(* IEC 61131-3 sources: Word/plc-course/24-capstone-projects/labs/starter, 3 files *)

(* ---- 24-1-conveyor-sorting-cell.st ---- *)
(* Capstone 24-1: Conveyor sorting cell SC-1.
   Module 24 (Capstone projects). STARTER - the interface is done for you.

   Everything the acceptance test (FAT) uses is declared here: the I/O, the
   HMI interface structure and the configuration. Do not rename any of it.
   Everything else is your design. Read the brief first:
     24-capstone-projects/24-1-conveyor-sorting-cell.md

   Suggested workflow:
     1. Add your own types (state enumeration, tracking record, ...) in a
        second TYPE block, and your function blocks (for example FB_Alarm,
        FB_Pusher, FB_Tracker) between the TYPE blocks and the PROGRAM.
     2. Replace the placeholder body of SortingCell with your logic.
     3. Run the FAT and work through it milestone by milestone (M1..M7):
          python3 tools/plctest.py my-work/24-1-conveyor-sorting-cell.st \
                  24-capstone-projects/labs/24-1-conveyor-sorting-cell.test

   Training exercise only. The emergency stop is read here as an ordinary
   input so that the program can react to it. On a real machine the
   emergency stop is a safety function: a safety relay or safety PLC
   removes power from the motor and the pusher valves directly, and the
   standard PLC only monitors it (Module 20). *)

TYPE
  (* ---- HMI interface: part of the specification, do not change ---- *)
  ST_CellCmd : STRUCT            (* HMI -> PLC. The HMI sets a bit, the PLC acts once and clears it *)
    Start        : BOOL;         (* start the cell (Auto) *)
    Stop         : BOOL;         (* normal stop, always obeyed *)
    Ack          : BOOL;         (* acknowledge all alarms *)
    Reset        : BOOL;         (* acknowledge and reset alarms whose cause has gone *)
    CyclePusherA : BOOL;         (* Manual: one supervised stroke of pusher A *)
    CyclePusherB : BOOL;         (* Manual: one supervised stroke of pusher B *)
    ClearCounts  : BOOL;         (* zero all six production counters *)
  END_STRUCT;

  ST_CellSts : STRUCT            (* PLC -> HMI, rewritten every scan *)
    State          : INT;        (* 1 STOPPED, 2 STARTING, 3 RUNNING, 4 FAULTED, 5 MANUAL *)
    Ready          : BOOL;       (* a Start now would be accepted *)
    LaneAFull      : BOOL;       (* debounced lane-full status *)
    LaneBFull      : BOOL;
    PartsInTransit : INT;        (* registered parts not yet delivered *)
    CountMetal     : DINT;       (* classified at the entry station *)
    CountPlastic   : DINT;
    CountOversize  : DINT;
    CountLaneA     : DINT;       (* delivered, counted by the delivery eyes *)
    CountLaneB     : DINT;
    CountReject    : DINT;
  END_STRUCT;

  ST_CellAlm : STRUCT            (* PLC -> HMI. TRUE from detection until a successful reset *)
    EStop         : BOOL;
    MotorOverload : BOOL;
    EntryJam      : BOOL;        (* entry eye blocked too long *)
    Jam           : BOOL;        (* a part did not reach its delivery eye in time *)
    PusherA       : BOOL;        (* pusher A did not extend / retract / stay home *)
    PusherB       : BOOL;
    TrackOverflow : BOOL;        (* more parts on the belt than the tracking table holds *)
    Unacked       : BOOL;        (* at least one alarm not yet acknowledged *)
  END_STRUCT;

  ST_CellCfg : STRUCT            (* engineer settings; the defaults are the commissioning values *)
    StartWarnTime : TIME := T#3s;    (* horn before the belt moves (never less than 2 s) *)
    DistA         : INT  := 500;     (* mm from registration to pusher A *)
    DistB         : INT  := 1000;    (* mm from registration to pusher B *)
    JamTimeA      : TIME := T#3s;    (* running time allowed from registration to LaneA_PE *)
    JamTimeB      : TIME := T#4s;    (* ... to LaneB_PE *)
    JamTimeR      : TIME := T#5s;    (* ... to RejectPE *)
    EntryJamTime  : TIME := T#2s;    (* entry eye blocked while running *)
    PusherTimeout : TIME := T#1s;    (* each pusher movement must finish within this *)
    LaneFullTime  : TIME := T#1s;    (* lane-full eye debounce, on and off *)
  END_STRUCT;

  ST_CellHmi : STRUCT
    Cmd : ST_CellCmd;
    Sts : ST_CellSts;
    Alm : ST_CellAlm;
    Cfg : ST_CellCfg;
  END_STRUCT;
END_TYPE

(* TODO: your own TYPE block and your function blocks go here. *)

PROGRAM SortingCell
  VAR (* operator panel *)
    StartPB    AT %IX0.0 : BOOL;   (* Start, NO *)
    StopPB_NC  AT %IX0.1 : BOOL;   (* Stop, NC: TRUE while not pressed *)
    EStop_NC   AT %IX0.2 : BOOL;   (* e-stop circuit monitoring, NC: TRUE while healthy *)
    ResetPB    AT %IX0.3 : BOOL;   (* Reset, NO *)
    ModeAuto   AT %IX0.4 : BOOL;   (* mode selector in AUTO *)
    ModeManual AT %IX0.5 : BOOL;   (* mode selector in MAN *)
    JogPB      AT %IX0.6 : BOOL;   (* Jog forward, NO, hold-to-run *)
    MotorOL_NC AT %IX0.7 : BOOL;   (* conveyor motor overload relay, NC: TRUE while healthy *)
  END_VAR
  VAR (* conveyor sensors *)
    EntryPE       AT %IX1.0 : BOOL;  (* entry eye: TRUE while a part blocks it *)
    MetalPX       AT %IX1.1 : BOOL;  (* inductive sensor: TRUE = metal *)
    TallPE        AT %IX1.2 : BOOL;  (* height eye: TRUE = part too tall *)
    LaneA_PE      AT %IX1.3 : BOOL;  (* lane A delivery eye *)
    LaneB_PE      AT %IX1.4 : BOOL;  (* lane B delivery eye *)
    RejectPE      AT %IX1.5 : BOOL;  (* reject chute eye *)
    LaneA_FullPE  AT %IX1.6 : BOOL;  (* lane A full eye: TRUE = blocked *)
    LaneB_FullPE  AT %IX1.7 : BOOL;  (* lane B full eye *)
    PusherA_ExtLS AT %IX2.0 : BOOL;  (* pusher A extended *)
    PusherA_RetLS AT %IX2.1 : BOOL;  (* pusher A retracted (home) *)
    PusherB_ExtLS AT %IX2.2 : BOOL;  (* pusher B extended *)
    PusherB_RetLS AT %IX2.3 : BOOL;  (* pusher B retracted (home) *)
    EncCount      AT %IW0 : UINT;    (* belt encoder via high-speed counter: 1 count = 1 mm *)
  END_VAR
  VAR (* outputs *)
    ConveyorRun AT %QX0.0 : BOOL;    (* conveyor motor contactor *)
    PusherA_Sol AT %QX0.1 : BOOL;    (* pusher A solenoid valve: TRUE = extend *)
    PusherB_Sol AT %QX0.2 : BOOL;    (* pusher B solenoid valve *)
    Horn        AT %QX0.3 : BOOL;    (* start-up warning horn *)
    GreenLamp   AT %QX0.4 : BOOL;    (* stack light green: running *)
    AmberLamp   AT %QX0.5 : BOOL;    (* stack light amber: lane full *)
    RedLamp     AT %QX0.6 : BOOL;    (* stack light red: alarm *)
  END_VAR
  VAR (* HMI interface *)
    HMI : ST_CellHmi;
  END_VAR
  (* TODO: your internal variables and function block instances. *)

  (* TODO: replace these placeholder lines with the cell logic.
     (MATIEC needs at least one statement in a program body.) *)
  ConveyorRun := FALSE;
  PusherA_Sol := FALSE;
  PusherB_Sol := FALSE;
  Horn := FALSE;
  GreenLamp := FALSE;
  AmberLamp := FALSE;
  RedLamp := FALSE;
  HMI.Sts.State := 1;
END_PROGRAM

CONFIGURATION Config0
  RESOURCE Res0 ON PLC
    TASK MainTask(INTERVAL := T#10ms, PRIORITY := 0);
    PROGRAM Inst0 WITH MainTask : SortingCell;
  END_RESOURCE
END_CONFIGURATION

(* ---- 24-2-batch-mixing-plant.st ---- *)
(* Capstone 24-2: Batch mixing plant (mixing vessel T-201).
   Module 24 (Capstone projects). STARTER - the interface, the recipe,
   configuration, HMI and report data types, and the plant simulation are
   done for you. Write the control logic where it says TODO (add your own
   functions, function blocks and variables as you wish), then run:
     python3 tools/plctest.py 24-capstone-projects/labs/starter/24-2-batch-mixing-plant.st
   Brief: 24-capstone-projects/24-2-batch-mixing-plant.md *)

(* =====================================================================
   GIVEN TYPES - part of the project interface. Do not change them: the
   acceptance test and the HMI depend on these names.
   ===================================================================== *)
TYPE
  (* Procedural state of the batch (a subset of the ISA-88 state model).
     Holding, Restarting and Aborting are transient: the batch passes
     through them while their actions complete. *)
  E_BatchState : (Idle, Running, Holding, Held, Restarting, Aborting,
                  Aborted, Complete);

  (* Phase of the batch procedure that is active, or was active when the
     batch was held. PhaseNone when no batch is in progress. *)
  E_BatchPhase : (PhaseNone, PhaseChargeA, PhaseChargeB, PhaseHeat,
                  PhaseMix, PhaseDrain);

  (* One recipe (the ISA-88 "formula": the parameters of the procedure) *)
  ST_Recipe : STRUCT
    Name     : STRING;    (* shown on the HMI and in the batch report *)
    QtyA     : REAL;      (* ingredient A to charge, litres *)
    QtyB     : REAL;      (* ingredient B to charge, litres; 0.0 = none *)
    TempSP   : REAL;      (* process temperature setpoint, degC *)
    MixTime  : TIME;      (* minimum agitation time in the mix/hold phase *)
    HoldTime : TIME;      (* time the contents must spend at temperature *)
  END_STRUCT;

  (* Engineering configuration. The defaults suit the plant; the test
     changes a few of them to check that your program uses them. *)
  ST_BatchCfg : STRUCT
    LitresPerPulseA : REAL := 0.5;    (* FT-201 K-factor: 2 pulses per litre *)
    LitresPerPulseB : REAL := 0.1;    (* FT-202 K-factor: 10 pulses per litre *)
    PreactA         : REAL := 4.0;    (* in-flight volume of XV-201, L: close this early *)
    PreactB         : REAL := 1.0;    (* in-flight volume of XV-202, L *)
    SettleTime      : TIME := T#3s;   (* after an inlet closes, before the charge is complete *)
    NoFlowTime      : TIME := T#10s;  (* inlet open, no meter pulse for this long = dosing fault *)
    MaxChargeTime   : TIME := T#5m;   (* longest a charge phase may run = dosing fault *)
    MaxHeatTime     : TIME := T#15m;  (* longest the heating phase may run = heating timeout *)
    TempBand        : REAL := 2.0;    (* "at temperature" = within +/- this of TempSP, degC *)
    TempHighLimit   : REAL := 85.0;   (* high temperature alarm, degC (clears 2 degC below) *)
    TempKc          : REAL := 8.0;    (* TIC-203 gain, % per degC (ideal form) *)
    TempTi          : REAL := 200.0;  (* TIC-203 integral time, s *)
    TempTd          : REAL := 0.0;    (* TIC-203 derivative time, s *)
    AgitStartLevel  : REAL := 10.0;   (* agitator may start at or above this level, % *)
    AgitStopLevel   : REAL := 8.0;    (* agitator stops below this level, % *)
    HeatMinLevel    : REAL := 12.0;   (* heating allowed at or above this level, % *)
    EmptyLevel      : REAL := 1.0;    (* vessel empty at or below this level, % *)
    DrainRunOn      : TIME := T#5s;   (* pump keeps running this long after empty *)
    ValveLeadTime   : TIME := T#2s;   (* XV-204 opens this long before P-204 starts,
                                         and closes this long after it stops *)
    FeedbackTime    : TIME := T#3s;   (* motor command/feedback disagreement = fault *)
    XmtrFaultDelay  : TIME := T#2s;   (* NE43 failure must persist this long *)
    MinBatchL       : REAL := 300.0;  (* smallest valid batch (QtyA + QtyB), L *)
    MaxBatchL       : REAL := 1500.0; (* largest valid batch, L *)
    MinTempSP       : REAL := 20.0;   (* lowest valid recipe setpoint, degC (no cooling) *)
    MaxTempSP       : REAL := 80.0;   (* highest valid recipe setpoint, degC *)
  END_STRUCT;

  (* HMI interface. Commands: the HMI sets them TRUE, the PLC acts on them
     once and clears them in the same scan. Status: written by the PLC. *)
  ST_BatchHmi : STRUCT
    CmdStart     : BOOL;          (* start a batch with recipe RecipeNo *)
    CmdHold      : BOOL;
    CmdRestart   : BOOL;
    CmdAbort     : BOOL;
    CmdReset     : BOOL;          (* reset faults; Complete/Aborted -> Idle *)
    CmdAck       : BOOL;          (* acknowledge all alarms *)
    CmdDrain     : BOOL;          (* empty the vessel (from Idle only) *)
    RecipeNo     : INT := 1;      (* operator's recipe selection, 1..5 *)
    State        : E_BatchState;
    Phase        : E_BatchPhase;
    ActiveRecipe : INT;           (* recipe of the batch in progress; 0 = none *)
    RejectCode   : INT;           (* result of the last Start: 0 = accepted *)
    LevelPct     : REAL;          (* LT-201, % *)
    TempC        : REAL;          (* TT-203, degC *)
    TotalA       : REAL;          (* ingredient A counted this batch, L *)
    TotalB       : REAL;          (* ingredient B counted this batch, L *)
    AlmActive    : WORD;          (* one bit per alarm, see the brief *)
    AlmUnack     : WORD;          (* same bits: not yet acknowledged *)
  END_STRUCT;

  (* Written once per completed batch (quality record) *)
  ST_BatchReport : STRUCT
    BatchCount : DINT;            (* batches completed since power-up *)
    RecipeNo   : INT;
    RecipeName : STRING;
    ActualA    : REAL;            (* litres counted by FT-201, in-flight included *)
    ActualB    : REAL;            (* litres counted by FT-202 *)
    BatchTime  : TIME;            (* Start accepted -> Complete, time held included *)
    MaxTemp    : REAL;            (* highest TT-203 reading during the batch, degC *)
  END_STRUCT;
END_TYPE

(* =====================================================================
   GIVEN PLANT SIMULATION - do not change.
   FB_PlantSim models the vessel, its valves, motors and instruments well
   enough to test the control logic. It also records "observer" values
   that the acceptance test uses as an independent referee (for example,
   how many litres really went into the vessel, whatever your program
   counted).

   The program calls it once per scan with last scan's outputs and copies
   its outputs into the input image. The test drives it by writing its
   inputs (set Sim.FlowFactorA 0.0, set Sim.AgitatorFail TRUE, ...).

   Model (see the brief for more):
   - Vessel T-201: 2000 L = 100 %, flat bottom (1 % = 20 L).
   - XV-201, XV-202, XV-204: 2 s full stroke, spring-return (fail closed).
     Flow is proportional to the valve position.
   - Ingredient A: 4.0 L/s fully open; FT-201 gives one pulse per 0.5 L.
     Ingredient B: 1.0 L/s fully open; FT-202 gives one pulse per 0.1 L.
     Each pulse is a square wave (on for half the pulse volume).
   - P-204 pumps 6.0 L/s through a fully open XV-204; its flow falls away
     below 10 L in the vessel.
   - M-201 running feedback 1.0 s after its command, P-204 0.5 s; both
     drop at once when the command drops or the motor fails.
   - Heating: TV-203 (0..27648 counts = 0..100 %) admits steam to the
     jacket. The heat reaches the contents through a 10 s lag, is reduced
     as the contents approach the 130 degC steam temperature, and falls to
     30 % if the agitator is stopped. The vessel loses heat slowly to the
     20 degC surroundings. TT-203 sits in a thermowell (3 s lag).
     Ingredients enter at 20 degC.
   - LT-201 0..100 % and TT-203 0..150 degC are 4-20 mA transmitters
     (NE43: they saturate at 3.8 and 20.5 mA). The analog card reads
     4 mA = 0 and 20 mA = 27648 counts (1728 counts per mA) and clips at
     -4864 and 32511.
   - LSHH-201 trips at 1800 L (90 %) and resets at 1780 L. NC contact.
   - PowerOK FALSE (safety relay open) removes power from every field
     output: valves close, motors stop, the steam valve closes.
   - Physics is integrated in fixed 10 ms steps.
   ===================================================================== *)
FUNCTION_BLOCK FB_PlantSim
  VAR_INPUT
    InletA       : BOOL;           (* XV-201 open command *)
    InletB       : BOOL;           (* XV-202 open command *)
    Outlet       : BOOL;           (* XV-204 open command *)
    Agitator     : BOOL;           (* M-201 run command *)
    Pump         : BOOL;           (* P-204 run command *)
    HeatValveRaw : INT;            (* TV-203 analog output, counts *)
    PowerOK      : BOOL := TRUE;   (* safety relay closed *)
    (* fault injection and test hooks *)
    FlowFactorA  : REAL := 1.0;    (* supply A: 1.0 normal, 0.0 no flow, 0.3 partly blocked *)
    FlowFactorB  : REAL := 1.0;    (* supply B *)
    AgitatorFail : BOOL;           (* M-201 will not run (or trips if running) *)
    PumpFail     : BOOL;           (* P-204 will not run (or trips if running) *)
    HeatFail     : BOOL;           (* no steam: the jacket gives no heat *)
    HHWireBreak  : BOOL;           (* LSHH-201 circuit open *)
    TtForce      : BOOL;           (* TT-203 loop current replaced by TtForcemA *)
    TtForcemA    : REAL := 12.0;   (*   (a loop calibrator, or a failed loop) *)
    LtForce      : BOOL;           (* LT-201 loop current replaced by LtForcemA *)
    LtForcemA    : REAL := 12.0;
  END_VAR
  VAR_OUTPUT
    (* field signals, copied to the PLC input image *)
    FlowPulseA      : BOOL;
    FlowPulseB      : BOOL;
    AgitatorRunning : BOOL;
    PumpRunning     : BOOL;
    LevelHH_NC      : BOOL := TRUE;
    LevelRaw        : INT;
    TempRaw         : INT;
    (* process state: a test may SET these to jump to a new condition *)
    VolumeL         : LREAL := 0.0;   (* liquid in the vessel, L *)
    TempC           : REAL := 20.0;   (* true temperature of the contents, degC *)
    (* observer values, for the tests *)
    HeatValvePct    : REAL;           (* steam valve position the plant sees, % *)
    DeliveredA      : LREAL;          (* true litres through XV-201 since power-up *)
    DeliveredB      : LREAL;          (* true litres through XV-202 *)
    DrainedL        : LREAL;          (* true litres pumped out *)
    MaxVolumeL      : REAL;           (* highest volume seen *)
    MaxTempC        : REAL := 20.0;   (* highest true temperature seen (a test may reset it) *)
    AgitatorDryS    : REAL;           (* s the agitator ran with less than 150 L in the vessel *)
    HeatNoAgitS     : REAL;           (* s of steam with the agitator stopped or < 200 L *)
    DeadheadS       : REAL;           (* s P-204 ran without XV-204 fully open *)
  END_VAR
  VAR CONSTANT
    STEP_TIME     : TIME := T#10ms;   (* integration step *)
    STEP_S        : REAL := 0.01;
    VESSEL_L      : REAL := 2000.0;
    AMBIENT_C     : REAL := 20.0;
    STROKE_S      : REAL := 2.0;      (* valve full stroke *)
    FLOW_A_LPS    : REAL := 4.0;
    FLOW_B_LPS    : REAL := 1.0;
    PUMP_LPS      : REAL := 6.0;
    HALF_PULSE_A  : LREAL := 0.25;    (* half of 0.5 L per pulse *)
    HALF_PULSE_B  : LREAL := 0.05;    (* half of 0.1 L per pulse *)
    AGIT_START_S  : REAL := 1.0;
    PUMP_START_S  : REAL := 0.5;
    HEAT_DUTY     : REAL := 150.0;    (* L.degC/s at 100 % valve, cold contents *)
    STEAM_C       : REAL := 130.0;
    JACKET_TAU_S  : REAL := 10.0;
    WELL_TAU_S    : REAL := 3.0;
    LOSS_LPS      : REAL := 0.45;     (* heat loss coefficient, L/s *)
    HH_TRIP_L     : LREAL := 1800.0;
    HH_RESET_L    : LREAL := 1780.0;
  END_VAR
  VAR
    Clock : TON;
    LastET : TIME;
    DeltaT : TIME;
    StepAcc : TIME;
    PosA : REAL;
    PosB : REAL;
    PosOut : REAL;
    AgitAcc : REAL;
    PumpAcc : REAL;
    AgitOn : BOOL;
    PumpOn : BOOL;
    QA : REAL;
    QB : REAL;
    QOut : REAL;
    dA : LREAL;
    dB : LREAL;
    dOut : LREAL;
    VRest : LREAL;
    VNew : LREAL;
    PulseAccA : LREAL;
    PulseAccB : LREAL;
    PulseA : BOOL;
    PulseB : BOOL;
    HeatTarget : REAL;
    HeatFlow : REAL;
    VEff : REAL;
    WellC : REAL := 20.0;
    HHWet : BOOL;
    mA : REAL;
    Started : BOOL;
  END_VAR

  (* --- time since the previous call (IEC has no system clock function) --- *)
  Clock(IN := TRUE, PT := T#24h);
  DeltaT := SUB_TIME(Clock.ET, LastET);
  LastET := Clock.ET;
  IF Clock.Q THEN                 (* re-arm once a day *)
    Clock(IN := FALSE);
    LastET := T#0s;
  END_IF;
  IF NOT Started THEN
    Started := TRUE;
    WellC := TempC;
  END_IF;

  IF PowerOK THEN
    HeatValvePct := LIMIT(0.0, INT_TO_REAL(HeatValveRaw) * 100.0 / 27648.0, 100.0);
  ELSE
    HeatValvePct := 0.0;
  END_IF;

  StepAcc := ADD_TIME(StepAcc, DeltaT);
  WHILE StepAcc >= STEP_TIME DO
    StepAcc := SUB_TIME(StepAcc, STEP_TIME);

    (* --- valves: 2 s stroke, spring return --- *)
    IF InletA AND PowerOK THEN
      PosA := MIN(1.0, PosA + STEP_S / STROKE_S);
    ELSE
      PosA := MAX(0.0, PosA - STEP_S / STROKE_S);
    END_IF;
    IF InletB AND PowerOK THEN
      PosB := MIN(1.0, PosB + STEP_S / STROKE_S);
    ELSE
      PosB := MAX(0.0, PosB - STEP_S / STROKE_S);
    END_IF;
    IF Outlet AND PowerOK THEN
      PosOut := MIN(1.0, PosOut + STEP_S / STROKE_S);
    ELSE
      PosOut := MAX(0.0, PosOut - STEP_S / STROKE_S);
    END_IF;

    (* --- motors and their running feedback --- *)
    IF Agitator AND PowerOK AND NOT AgitatorFail THEN
      AgitAcc := MIN(AgitAcc + STEP_S, AGIT_START_S);
    ELSE
      AgitAcc := 0.0;
    END_IF;
    AgitOn := AgitAcc >= AGIT_START_S;
    IF Pump AND PowerOK AND NOT PumpFail THEN
      PumpAcc := MIN(PumpAcc + STEP_S, PUMP_START_S);
    ELSE
      PumpAcc := 0.0;
    END_IF;
    PumpOn := PumpAcc >= PUMP_START_S;

    (* --- flows, L/s, and volumes for this step --- *)
    QA := FLOW_A_LPS * PosA * LIMIT(0.0, FlowFactorA, 2.0);
    QB := FLOW_B_LPS * PosB * LIMIT(0.0, FlowFactorB, 2.0);
    IF PumpOn THEN
      QOut := PUMP_LPS * PosOut * LIMIT(0.0, LREAL_TO_REAL(VolumeL) / 10.0, 1.0);
    ELSE
      QOut := 0.0;
    END_IF;
    dA := REAL_TO_LREAL(QA * STEP_S);
    dB := REAL_TO_LREAL(QB * STEP_S);
    dOut := MIN(REAL_TO_LREAL(QOut * STEP_S), MAX(VolumeL, 0.0));

    (* --- mass balance; feeds enter at ambient temperature --- *)
    VRest := VolumeL - dOut;
    VNew := VRest + dA + dB;
    IF VNew > 0.001 THEN
      TempC := LREAL_TO_REAL((REAL_TO_LREAL(TempC) * VRest
                              + REAL_TO_LREAL(AMBIENT_C) * (dA + dB)) / VNew);
    END_IF;
    VolumeL := LIMIT(0.0, VNew, REAL_TO_LREAL(VESSEL_L));  (* full = overflow line *)
    DeliveredA := DeliveredA + dA;
    DeliveredB := DeliveredB + dB;
    DrainedL := DrainedL + dOut;

    (* --- flow meter pulses: toggle every half pulse volume --- *)
    PulseAccA := PulseAccA + dA;
    IF PulseAccA >= HALF_PULSE_A THEN
      PulseAccA := PulseAccA - HALF_PULSE_A;
      PulseA := NOT PulseA;
    END_IF;
    PulseAccB := PulseAccB + dB;
    IF PulseAccB >= HALF_PULSE_B THEN
      PulseAccB := PulseAccB - HALF_PULSE_B;
      PulseB := NOT PulseB;
    END_IF;

    (* --- heating: steam duty through the jacket lag --- *)
    IF HeatFail THEN
      HeatTarget := 0.0;
    ELSE
      HeatTarget := HEAT_DUTY * HeatValvePct / 100.0
                    * MAX(0.0, (STEAM_C - TempC) / (STEAM_C - AMBIENT_C));
      IF NOT AgitOn THEN
        HeatTarget := HeatTarget * 0.3;
      END_IF;
    END_IF;
    HeatFlow := HeatFlow + (HeatTarget - HeatFlow) * STEP_S / JACKET_TAU_S;
    VEff := MAX(LREAL_TO_REAL(VolumeL), 50.0);
    TempC := TempC + (HeatFlow - LOSS_LPS * (TempC - AMBIENT_C)) / VEff * STEP_S;
    WellC := WellC + (TempC - WellC) * STEP_S / WELL_TAU_S;

    (* --- observers --- *)
    IF AgitOn AND VolumeL < 150.0 THEN
      AgitatorDryS := AgitatorDryS + STEP_S;
    END_IF;
    IF HeatValvePct > 1.0 AND (NOT AgitOn OR VolumeL < 200.0) THEN
      HeatNoAgitS := HeatNoAgitS + STEP_S;
    END_IF;
    IF PumpOn AND PosOut < 0.99 THEN
      DeadheadS := DeadheadS + STEP_S;
    END_IF;
    MaxVolumeL := MAX(MaxVolumeL, LREAL_TO_REAL(VolumeL));
    MaxTempC := MAX(MaxTempC, TempC);
  END_WHILE;

  (* --- high-high level switch, NC: opens on high level or a broken wire --- *)
  IF VolumeL >= HH_TRIP_L THEN
    HHWet := TRUE;
  ELSIF VolumeL <= HH_RESET_L THEN
    HHWet := FALSE;
  END_IF;
  LevelHH_NC := NOT HHWet AND NOT HHWireBreak;

  (* --- transmitters and analog input card --- *)
  mA := LIMIT(3.8, 4.0 + 16.0 * LREAL_TO_REAL(VolumeL) / VESSEL_L, 20.5);
  IF LtForce THEN
    mA := LtForcemA;
  END_IF;
  LevelRaw := REAL_TO_INT(LIMIT(-4864.0, (mA - 4.0) * 1728.0, 32511.0));
  mA := LIMIT(3.8, 4.0 + 16.0 * WellC / 150.0, 20.5);
  IF TtForce THEN
    mA := TtForcemA;
  END_IF;
  TempRaw := REAL_TO_INT(LIMIT(-4864.0, (mA - 4.0) * 1728.0, 32511.0));

  (* --- outputs --- *)
  FlowPulseA := PulseA;
  FlowPulseB := PulseB;
  AgitatorRunning := AgitOn;
  PumpRunning := PumpOn;
END_FUNCTION_BLOCK

PROGRAM BatchMixer
  VAR (* digital inputs *)
    FlowPulseA      AT %IX0.0 : BOOL;  (* FT-201 ingredient A meter: one pulse per 0.5 L *)
    FlowPulseB      AT %IX0.1 : BOOL;  (* FT-202 ingredient B meter: one pulse per 0.1 L *)
    AgitatorRunning AT %IX0.2 : BOOL;  (* M-201 agitator running feedback (contactor aux) *)
    PumpRunning     AT %IX0.3 : BOOL;  (* P-204 drain pump running feedback *)
    LevelHH_NC      AT %IX0.4 : BOOL;  (* LSHH-201, NC: FALSE = high-high level or wire broken *)
    EStopOK_NC      AT %IX0.5 : BOOL;  (* safety relay status, NC: FALSE = e-stop operated *)
  END_VAR
  VAR (* analog inputs *)
    LevelRaw        AT %IW0 : INT;     (* LT-201 level 0-100 % (0-2000 L), 4 mA = 0, 20 mA = 27648 *)
    TempRaw         AT %IW1 : INT;     (* TT-203 temperature 0-150 degC, same card range *)
  END_VAR
  VAR (* digital outputs *)
    InletAValve     AT %QX0.0 : BOOL;  (* XV-201 ingredient A inlet valve, TRUE = open *)
    InletBValve     AT %QX0.1 : BOOL;  (* XV-202 ingredient B inlet valve *)
    OutletValve     AT %QX0.2 : BOOL;  (* XV-204 outlet valve *)
    AgitatorRun     AT %QX0.3 : BOOL;  (* M-201 agitator contactor *)
    PumpRun         AT %QX0.4 : BOOL;  (* P-204 drain pump contactor *)
    AlarmHorn       AT %QX0.5 : BOOL;  (* ON while any alarm is unacknowledged *)
    AlarmLamp       AT %QX0.6 : BOOL;  (* ON while any alarm is active *)
  END_VAR
  VAR (* analog output *)
    HeatValveRaw    AT %QW0 : INT;     (* TV-203 steam valve, 0 = closed .. 27648 = fully open *)
  END_VAR
  VAR RETAIN (* recipes and configuration survive a power cycle *)
    Recipes : ARRAY[1..5] OF ST_Recipe := [
      (Name := 'Floor cleaner', QtyA := 400.0, QtyB := 50.0, TempSP := 60.0,
       MixTime := T#60s, HoldTime := T#90s),
      (Name := 'Degreaser', QtyA := 250.0, QtyB := 120.0, TempSP := 45.0,
       MixTime := T#120s, HoldTime := T#30s),
      (Name := 'Cold blend', QtyA := 260.0, QtyB := 40.0, TempSP := 20.0,
       MixTime := T#30s, HoldTime := T#0s)];   (* recipes 4 and 5 are empty *)
    Cfg : ST_BatchCfg;
  END_VAR
  VAR (* given *)
    Hmi : ST_BatchHmi;                 (* HMI interface *)
    Report : ST_BatchReport;           (* last completed batch *)
    Sim : FB_PlantSim;                 (* plant simulation *)
    SimEnable : BOOL := TRUE;          (* set FALSE (or delete section 1) on a real PLC *)
  END_VAR

  (* ===== 1. PLANT SIMULATION (given - do not change) ====================
     The simulation plays the part of the field: it reads last scan's
     outputs and writes this scan's input image, just as the I/O system
     would. EStopOK_NC is a real input (the test sets it); the simulation
     only uses it to cut power to the field outputs, as the safety relay
     would. On a real PLC this section is removed and nothing else changes. *)
  IF SimEnable THEN
    Sim(InletA := InletAValve, InletB := InletBValve, Outlet := OutletValve,
        Agitator := AgitatorRun, Pump := PumpRun, HeatValveRaw := HeatValveRaw,
        PowerOK := EStopOK_NC);
    FlowPulseA := Sim.FlowPulseA;
    FlowPulseB := Sim.FlowPulseB;
    AgitatorRunning := Sim.AgitatorRunning;
    PumpRunning := Sim.PumpRunning;
    LevelHH_NC := Sim.LevelHH_NC;
    LevelRaw := Sim.LevelRaw;
    TempRaw := Sim.TempRaw;
  END_IF;

  (* ===== 2. YOUR CONTROL LOGIC ==========================================
     TODO: replace the placeholder lines below. A suggested layout (see
     "Suggested architecture" in the brief):
       2. time base; HMI commands (latch them, then clear the Cmd bits)
       3. measurements: LT-201 and TT-203 scaling, NE43 checks, flow totals
       4. alarms and faults: detect, latch, reset, acknowledge
       5. batch state machine (Idle/Running/Holding/Held/...) and the
          phase sequence (ChargeA -> ChargeB -> Heat -> Mix -> Drain)
       6. equipment control: inlet dosing, agitator, TIC-203 PID and
          steam valve, drain valve and pump, all with their interlocks
       7. outputs, e-stop override, HMI status and the batch report
     Keep the names in the brief's interface tables: the acceptance test
     uses them. *)
  InletAValve := FALSE;
  InletBValve := FALSE;
  OutletValve := FALSE;
  AgitatorRun := FALSE;
  PumpRun := FALSE;
  HeatValveRaw := 0;
  AlarmHorn := FALSE;
  AlarmLamp := FALSE;
  Hmi.State := Idle;
END_PROGRAM

CONFIGURATION Config0
  RESOURCE Res0 ON PLC
    TASK MainTask(INTERVAL := T#10ms, PRIORITY := 0);
    PROGRAM Inst0 WITH MainTask : BatchMixer;
  END_RESOURCE
END_CONFIGURATION

(* ---- 24-3-pump-station.st ---- *)
(* Capstone 24-3: Wastewater pump station (wet-well lift station).
   Module 24 (Capstone projects). STARTER - the interface, the SCADA data
   types and the plant simulation are done for you. Write the control
   logic where it says TODO (add your own functions, function blocks and
   variables as you wish), then run:
     python3 tools/plctest.py 24-capstone-projects/labs/starter/24-3-pump-station.st
   Brief: 24-capstone-projects/24-3-pump-station.md *)

(* =====================================================================
   GIVEN TYPES - part of the project interface. Do not change them: the
   acceptance test and the SCADA register map depend on these names.
   ===================================================================== *)
TYPE
  (* Fault injection for the simulated level transmitter *)
  E_XmtrFault : (XmtrOK,          (* healthy: 4-20 mA follows the level  *)
                 XmtrWireBreak,   (* loop open: 0 mA                     *)
                 XmtrLow,         (* failed downscale: 3.5 mA            *)
                 XmtrHigh,        (* failed upscale: 21.5 mA             *)
                 XmtrFrozen);     (* output stuck at its present value   *)

  (* Setpoints. SCADA writes these (holding registers 40101-40108). The
     levels are integers in millimetres above the wet-well floor. *)
  ST_Config : STRUCT
    DutyStartMm      : INT := 1500;   (* lead pump starts at or above       *)
    DutyStopMm       : INT := 600;    (* lead pump stops at or below        *)
    AssistStartMm    : INT := 1900;   (* assist pump starts at or above     *)
    AssistStopMm     : INT := 900;    (* assist pump stops at or below      *)
    HighAlarmMm      : INT := 2200;   (* high-level alarm                   *)
    LowAlarmMm       : INT := 450;    (* low-level alarm and dry-run cut-out *)
    MaxStartsPerHour : INT := 6;      (* per pump, rolling 60 min; 0 = off  *)
    BalanceByHours   : BOOL := FALSE; (* FALSE = rotate lead each cycle,
                                         TRUE = lead = least run time      *)
  END_STRUCT;

  (* One pump in the SCADA interface (4 registers + 2 x 32-bit values) *)
  ST_PumpScada : STRUCT
    Status         : WORD;  (* bit 0 in Auto, 1 available, 2 run command,
                               3 running, 4 overload fault, 5 feedback fault,
                               6 start-limited *)
    Starts         : DINT;  (* total starts (rising edges of the running feedback) *)
    RunSeconds     : DINT;  (* total running time, s *)
    StartsLastHour : INT;   (* starts in the last 60 minutes *)
  END_STRUCT;

  (* The whole SCADA interface image *)
  ST_Scada : STRUCT
    StationStatus : WORD;   (* bit 0 level control, 1 float backup, 2 pumping,
                               3 any alarm active, 4 any alarm unacknowledged *)
    AlmActive     : WORD;   (* one bit per alarm, see the brief *)
    AlmUnack      : WORD;   (* same bits: alarm not yet acknowledged *)
    LevelMm       : INT;    (* measured level, mm (0-4000) *)
    LeadPump      : INT;    (* 1-3: pump that leads this cycle / the next cycle *)
    PumpsRunning  : INT;    (* number of running feedbacks *)
    Pump          : ARRAY[1..3] OF ST_PumpScada;
    CmdAck        : BOOL;   (* SCADA command: acknowledge alarms (PLC clears it) *)
    CmdReset      : BOOL;   (* SCADA command: reset faults (PLC clears it) *)
  END_STRUCT;
END_TYPE

(* =====================================================================
   GIVEN PLANT SIMULATION - do not change.
   FB_WetWellSim models the wet well, the three pumps and the level
   instruments well enough to test the control logic. It also records
   "observer" statistics that the acceptance test uses as an independent
   referee (for example, did any pump ever run dry?).

   The program calls it once per scan with the pump run commands, and
   copies its outputs into the input image. The test drives it by writing
   its inputs directly (set Sim.InflowLps 20.0, set Sim.Trip2 TRUE, ...).

   Model:
   - Wet well plan area 4.0 m2, so 1 m of level = 4000 L (1 cm = 40 L).
   - Level transmitter 0-4.00 m = 4-20 mA. The analog card reads
     4 mA = 0 and 20 mA = 27648 counts (1728 counts per mA) and clips at
     -4864 and 32511. A healthy transmitter stays within 3.8-20.5 mA.
   - Floats (with 5 cm switching differential):
       low float    wet at >= 0.40 m, dry at <= 0.35 m
       high float   trips at >= 2.50 m, resets at <= 2.45 m (NC contact)
       HH float     trips at >= 2.80 m, resets at <= 2.75 m (NC contact)
   - Station outflow: 1 pump 25 L/s, 2 pumps 40 L/s, 3 pumps 48 L/s
     (the rising main limits parallel pumping). The flow falls to zero as
     the level drops from 0.25 m (minimum submergence) to 0.10 m.
   - A pump gives its running feedback 0.5 s after its run command, unless
     it is tripped (TripN) or will not run (NoRunN). The feedback drops as
     soon as the command drops or the pump trips.
   - Above 3.20 m the well spills to the emergency overflow.
   - The level is integrated in fixed 0.1 s steps, independent of the
     task interval.
   ===================================================================== *)
FUNCTION_BLOCK FB_WetWellSim
  VAR_INPUT
    Run1 : BOOL;                 (* run commands from the PLC outputs *)
    Run2 : BOOL;
    Run3 : BOOL;
    InflowLps : REAL := 0.0;     (* sewage inflow to the well, L/s *)
    Trip1 : BOOL;                (* fault injection: overload relay tripped *)
    Trip2 : BOOL;
    Trip3 : BOOL;
    NoRun1 : BOOL;               (* fault injection: pump will not run and *)
    NoRun2 : BOOL;               (* gives no feedback (e.g. contactor coil  *)
    NoRun3 : BOOL;               (* open circuit)                           *)
    XmtrFault : E_XmtrFault := XmtrOK;  (* fault injection: transmitter *)
  END_VAR
  VAR_OUTPUT
    (* field signals, copied to the PLC input image *)
    LevelRaw : INT;              (* analog input, counts *)
    LowFloatWet : BOOL;          (* TRUE = low float submerged *)
    HighFloat_NC : BOOL := TRUE; (* FALSE = high float tripped *)
    HHFloat_NC : BOOL := TRUE;   (* FALSE = high-high float tripped *)
    Running1 : BOOL;             (* running feedbacks *)
    Running2 : BOOL;
    Running3 : BOOL;
    OverloadOK1_NC : BOOL := TRUE;  (* FALSE = overload tripped *)
    OverloadOK2_NC : BOOL := TRUE;
    OverloadOK3_NC : BOOL := TRUE;
    (* process state: a test may SET Level to jump to a new level *)
    Level : REAL := 1.0;         (* true level above the well floor, m *)
    OutflowLps : REAL;           (* pumped flow, L/s *)
    (* observer statistics, for the tests *)
    PumpsRunning : INT;          (* pumps running now *)
    MaxPumpsRunning : INT;       (* most pumps ever running together *)
    Starts1 : DINT;              (* starts seen per pump *)
    Starts2 : DINT;
    Starts3 : DINT;
    MaxStartsInHour : INT;       (* most starts of one pump in any 60 min *)
    DryRunS : REAL;              (* s that a pump ran below 0.25 m *)
    SpillL : REAL;               (* litres spilled to the overflow *)
    MinLevel : REAL;             (* lowest and highest true level seen *)
    MaxLevel : REAL;
  END_VAR
  VAR CONSTANT
    AREA_M2 : REAL := 4.0;
    SPAN_M : REAL := 4.0;
    COUNTS_PER_MA : REAL := 1728.0;
    OVERFLOW_M : REAL := 3.20;
    SUBMERGENCE_M : REAL := 0.25;
    SUCTION_M : REAL := 0.10;
    LOW_WET_M : REAL := 0.40;
    LOW_DRY_M : REAL := 0.35;
    HIGH_TRIP_M : REAL := 2.50;
    HIGH_RESET_M : REAL := 2.45;
    HH_TRIP_M : REAL := 2.80;
    HH_RESET_M : REAL := 2.75;
    STEP_TIME : TIME := T#100ms;
    STEP_S : REAL := 0.1;
    START_DELAY : TIME := T#500ms;
    HOUR_STEPS : DINT := 36000;  (* 60 min in 0.1 s steps *)
  END_VAR
  VAR
    Clock : TON;
    LastET : TIME;
    DeltaT : TIME;
    StepAcc : TIME;
    Steps : DINT;
    Started : BOOL;
    Cmd : ARRAY[1..3] OF BOOL;
    Trip : ARRAY[1..3] OF BOOL;
    NoRun : ARRAY[1..3] OF BOOL;
    Runs : ARRAY[1..3] OF BOOL;
    WasRunning : ARRAY[1..3] OF BOOL;
    StartAcc : ARRAY[1..3] OF TIME;
    StartCount : ARRAY[1..3] OF DINT;
    StartStamp : ARRAY[1..3, 0..31] OF DINT;
    NextStamp : ARRAY[1..3] OF INT;
    Flow : REAL;
    mA : REAL;
    HeldmA : REAL;
    i : INT;
    k : INT;
    n : INT;
    InHour : INT;
  END_VAR

  (* --- time since the previous call (IEC has no system clock function) --- *)
  Clock(IN := TRUE, PT := T#24h);
  DeltaT := SUB_TIME(Clock.ET, LastET);
  LastET := Clock.ET;
  IF Clock.Q THEN                 (* re-arm once a day *)
    Clock(IN := FALSE);
    LastET := T#0s;
  END_IF;
  IF NOT Started THEN
    Started := TRUE;
    MinLevel := Level;
    MaxLevel := Level;
    HeldmA := 4.0 + 16.0 * Level / SPAN_M;
  END_IF;

  Cmd[1] := Run1;    Cmd[2] := Run2;    Cmd[3] := Run3;
  Trip[1] := Trip1;  Trip[2] := Trip2;  Trip[3] := Trip3;
  NoRun[1] := NoRun1; NoRun[2] := NoRun2; NoRun[3] := NoRun3;

  (* --- pumps and their feedback --- *)
  n := 0;
  FOR i := 1 TO 3 DO
    IF Cmd[i] AND NOT Trip[i] AND NOT NoRun[i] THEN
      IF StartAcc[i] < START_DELAY THEN
        StartAcc[i] := ADD_TIME(StartAcc[i], DeltaT);
      END_IF;
    ELSE
      StartAcc[i] := T#0s;
    END_IF;
    Runs[i] := StartAcc[i] >= START_DELAY;
    IF Runs[i] THEN
      n := n + 1;
    END_IF;
    IF Runs[i] AND NOT WasRunning[i] THEN
      (* observer: count the start and the starts in the last 60 min *)
      StartCount[i] := StartCount[i] + 1;
      StartStamp[i, NextStamp[i]] := Steps;
      NextStamp[i] := (NextStamp[i] + 1) MOD 32;
      InHour := 0;
      FOR k := 0 TO 31 DO
        IF INT_TO_DINT(k) < StartCount[i] AND Steps - StartStamp[i, k] < HOUR_STEPS THEN
          InHour := InHour + 1;
        END_IF;
      END_FOR;
      MaxStartsInHour := MAX(MaxStartsInHour, InHour);
    END_IF;
    WasRunning[i] := Runs[i];
  END_FOR;
  PumpsRunning := n;
  MaxPumpsRunning := MAX(MaxPumpsRunning, n);

  (* --- wet-well level, fixed 0.1 s integration steps --- *)
  StepAcc := ADD_TIME(StepAcc, DeltaT);
  WHILE StepAcc >= STEP_TIME DO
    StepAcc := SUB_TIME(StepAcc, STEP_TIME);
    Steps := Steps + 1;
    CASE n OF
      0: Flow := 0.0;
      1: Flow := 25.0;
      2: Flow := 40.0;
    ELSE
      Flow := 48.0;
    END_CASE;
    Flow := Flow * LIMIT(0.0, (Level - SUCTION_M) / (SUBMERGENCE_M - SUCTION_M), 1.0);
    Level := Level + (InflowLps - Flow) * STEP_S / (1000.0 * AREA_M2);
    IF Level > OVERFLOW_M THEN
      SpillL := SpillL + (Level - OVERFLOW_M) * AREA_M2 * 1000.0;
      Level := OVERFLOW_M;
    ELSIF Level < 0.0 THEN
      Level := 0.0;
    END_IF;
    IF n > 0 AND Level < SUBMERGENCE_M THEN
      DryRunS := DryRunS + STEP_S;
    END_IF;
    MinLevel := MIN(MinLevel, Level);
    MaxLevel := MAX(MaxLevel, Level);
  END_WHILE;
  OutflowLps := Flow;

  (* --- floats --- *)
  IF Level >= LOW_WET_M THEN
    LowFloatWet := TRUE;
  ELSIF Level <= LOW_DRY_M THEN
    LowFloatWet := FALSE;
  END_IF;
  IF Level >= HIGH_TRIP_M THEN
    HighFloat_NC := FALSE;
  ELSIF Level <= HIGH_RESET_M THEN
    HighFloat_NC := TRUE;
  END_IF;
  IF Level >= HH_TRIP_M THEN
    HHFloat_NC := FALSE;
  ELSIF Level <= HH_RESET_M THEN
    HHFloat_NC := TRUE;
  END_IF;

  (* --- level transmitter and analog input card --- *)
  mA := LIMIT(3.8, 4.0 + 16.0 * Level / SPAN_M, 20.5);
  CASE XmtrFault OF
    XmtrWireBreak: mA := 0.0;
    XmtrLow:       mA := 3.5;
    XmtrHigh:      mA := 21.5;
    XmtrFrozen:    mA := HeldmA;
  END_CASE;
  HeldmA := mA;
  LevelRaw := REAL_TO_INT(LIMIT(-4864.0, (mA - 4.0) * COUNTS_PER_MA, 32511.0));

  (* --- outputs --- *)
  Running1 := Runs[1];
  Running2 := Runs[2];
  Running3 := Runs[3];
  OverloadOK1_NC := NOT Trip1;
  OverloadOK2_NC := NOT Trip2;
  OverloadOK3_NC := NOT Trip3;
  Starts1 := StartCount[1];
  Starts2 := StartCount[2];
  Starts3 := StartCount[3];
END_FUNCTION_BLOCK

PROGRAM PumpStation
  VAR (* digital inputs - station *)
    LowFloatWet        AT %IX0.0 : BOOL;  (* low float: TRUE = submerged (wet) *)
    HighFloat_NC       AT %IX0.1 : BOOL;  (* high float, NC: FALSE = >= 2.50 m or wire broken *)
    HHFloat_NC         AT %IX0.2 : BOOL;  (* high-high float, NC: FALSE = >= 2.80 m or broken *)
    AckPB              AT %IX0.3 : BOOL;  (* panel push-button: acknowledge alarms *)
    ResetPB            AT %IX0.4 : BOOL;  (* panel push-button: reset faults *)
  END_VAR
  VAR (* digital inputs - pumps *)
    Pump1Auto          AT %IX1.0 : BOOL;  (* Hand-Off-Auto switch in Auto *)
    Pump1Running       AT %IX1.1 : BOOL;  (* running feedback (contactor aux / VFD running relay) *)
    Pump1OverloadOK_NC AT %IX1.2 : BOOL;  (* motor protection healthy, NC: FALSE = tripped *)
    Pump2Auto          AT %IX2.0 : BOOL;
    Pump2Running       AT %IX2.1 : BOOL;
    Pump2OverloadOK_NC AT %IX2.2 : BOOL;
    Pump3Auto          AT %IX3.0 : BOOL;
    Pump3Running       AT %IX3.1 : BOOL;
    Pump3OverloadOK_NC AT %IX3.2 : BOOL;
  END_VAR
  VAR (* analog input *)
    LevelRaw           AT %IW0   : INT;   (* level transmitter 0-4.00 m, 4 mA = 0, 20 mA = 27648 *)
  END_VAR
  VAR (* digital outputs *)
    Pump1Run           AT %QX0.0 : BOOL;  (* run command to starter / VFD *)
    Pump2Run           AT %QX0.1 : BOOL;
    Pump3Run           AT %QX0.2 : BOOL;
    AlarmBeacon        AT %QX0.3 : BOOL;  (* flashing = unacknowledged, steady = active *)
  END_VAR
  VAR RETAIN (* setpoints survive a power cycle *)
    Cfg : ST_Config;                      (* written by SCADA *)
  END_VAR
  VAR (* given *)
    Scada : ST_Scada;                     (* SCADA interface image *)
    Sim : FB_WetWellSim;                  (* plant simulation *)
    SimEnable : BOOL := TRUE;             (* set FALSE (or delete section 1) on a real PLC *)
  END_VAR

  (* ===== 1. PLANT SIMULATION (given - do not change) ====================
     The simulation plays the part of the field: it reads last scan's
     outputs and writes this scan's input image, just as the I/O system
     would. On a real PLC this section is removed and nothing else changes. *)
  IF SimEnable THEN
    Sim(Run1 := Pump1Run, Run2 := Pump2Run, Run3 := Pump3Run);
    LevelRaw := Sim.LevelRaw;
    LowFloatWet := Sim.LowFloatWet;
    HighFloat_NC := Sim.HighFloat_NC;
    HHFloat_NC := Sim.HHFloat_NC;
    Pump1Running := Sim.Running1;
    Pump2Running := Sim.Running2;
    Pump3Running := Sim.Running3;
    Pump1OverloadOK_NC := Sim.OverloadOK1_NC;
    Pump2OverloadOK_NC := Sim.OverloadOK2_NC;
    Pump3OverloadOK_NC := Sim.OverloadOK3_NC;
  END_IF;

  (* ===== 2. YOUR CONTROL LOGIC ==========================================
     TODO: replace the placeholder lines below. A suggested layout (see
     "Suggested architecture" in the brief):
       2. time base and operator commands (AckPB, ResetPB, Scada.CmdAck,
          Scada.CmdReset - clear the SCADA command bits after use)
       3. level measurement: scaling, NE43 signal check, hold-last-good,
          float cross-check, latched transmitter fault -> float backup mode
       4. pump demand: duty / assist start-stop levels, float overrides,
          dry-run cut-out, never more than two pumps
       5. lead pump (rotation or run-time balancing), pump selection with
          start stagger and substitution, one pump block per pump
          (faults, availability, starts, run time, starts-per-hour)
       6. alarms: conditions -> AlmActive / AlmUnack, acknowledge, beacon
       7. SCADA image: status words, counters, level, lead pump
     Keep the variable names in the brief's interface tables: the
     acceptance test uses them. Read the plant only through the I/O
     variables, never through Sim.xxx: one FAT scenario switches the
     simulation off (SimEnable FALSE) and drives the inputs itself. *)
  Pump1Run := FALSE;
  Pump2Run := FALSE;
  Pump3Run := FALSE;
  AlarmBeacon := FALSE;
  Scada.LeadPump := 1;
END_PROGRAM

CONFIGURATION Config0
  RESOURCE Res0 ON PLC
    TASK MainTask(INTERVAL := T#10ms, PRIORITY := 0);
    PROGRAM Inst0 WITH MainTask : PumpStation;
  END_RESOURCE
END_CONFIGURATION
